FUNCTION_BLOCK MOTION_ACC_DCC
VAR_INPUT
	BOOL_UP_MOVE : BOOL;
	BOOL_DOWN_MOVE : BOOL;
	UINT_JOG_ACCDCC : UINT;
	UINT_HOME_ACCDCC : UINT;
	UINT_UD_ACCDCC : UINT;
	UINT_AG_ACCDCC : UINT;
	TIME_UD_DLY_ON : TIME;
	BOOL_MANUAL_PG : BOOL;
	BOOL_ORIGIN_COMP : BOOL;
	BOOL_ARM_HOME_READY : BOOL;
	STRING_CURRENT_PG : STRING;
	STRING_MAN_JOG_V_PG : STRING;
	STRING_MAN_POS_V_PG : STRING;
	STRING_MAN_JOG_H_PG : STRING;
	STRING_MAN_POS_H_PG : STRING;
END_VAR
VAR_OUTPUT

	UP_MOVE_ST_BOOL : BOOL;
	DOWN_MOVE_ST_BOOL : BOOL;
	ACC_UINT : UINT;
	DCC_UINT : UINT;

END_VAR
VAR
	T1: TON;
	T1COUNT: TIME;
	T2: TON;
	T2COUNT: TIME;
	MANJOGH: BOOL;
	MANJOGV: BOOL;
	MANPOSH: BOOL;
	MANPOSV: BOOL;
END_VAR
VAR // added by the converter: edge detectors and wires of the graphical bodies
    _w1, _w4, _w7, _w10 : BOOL;
    _w2, _w3, _w5, _w6, _w8, _w9, _w11, _w12 : UINT;
END_VAR

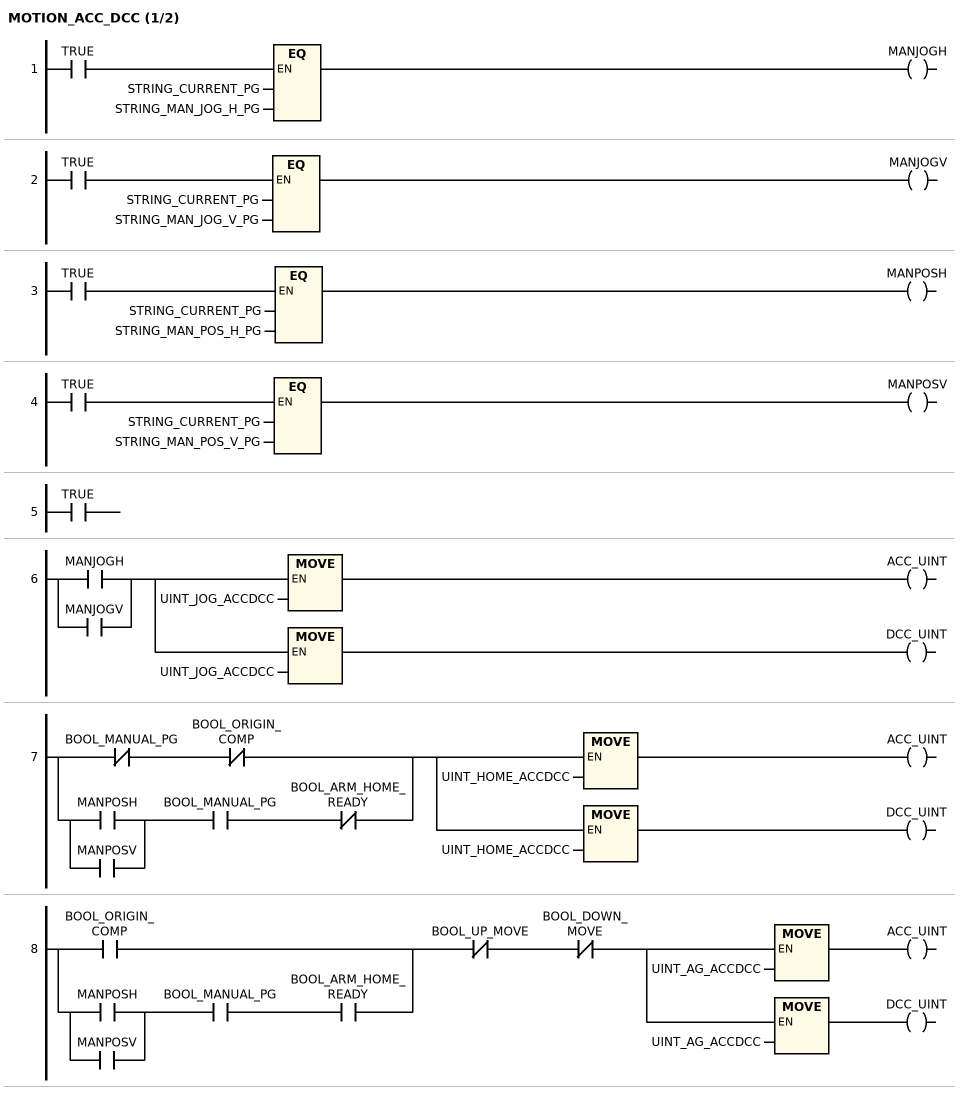
// NETWORK 1
MANJOGH := STRING_CURRENT_PG = STRING_MAN_JOG_H_PG;

// NETWORK 2
MANJOGV := STRING_CURRENT_PG = STRING_MAN_JOG_V_PG;

// NETWORK 3
MANPOSH := STRING_CURRENT_PG = STRING_MAN_POS_H_PG;

// NETWORK 4
MANPOSV := STRING_CURRENT_PG = STRING_MAN_POS_V_PG;

// NETWORK 5

// NETWORK 6
_w1 := MANJOGH OR MANJOGV;
IF _w1 THEN _w2 := UINT_JOG_ACCDCC; END_IF
ACC_UINT := _w2;
IF _w1 THEN _w3 := UINT_JOG_ACCDCC; END_IF
DCC_UINT := _w3;

// NETWORK 7
_w4 := NOT BOOL_MANUAL_PG AND NOT BOOL_ORIGIN_COMP OR (MANPOSH OR MANPOSV) AND BOOL_MANUAL_PG AND NOT BOOL_ARM_HOME_READY;
IF _w4 THEN _w5 := UINT_HOME_ACCDCC; END_IF
ACC_UINT := _w5;
IF _w4 THEN _w6 := UINT_HOME_ACCDCC; END_IF
DCC_UINT := _w6;

// NETWORK 8
_w7 := (BOOL_ORIGIN_COMP OR (MANPOSH OR MANPOSV) AND BOOL_MANUAL_PG AND BOOL_ARM_HOME_READY) AND NOT BOOL_UP_MOVE AND NOT BOOL_DOWN_MOVE;
IF _w7 THEN _w8 := UINT_AG_ACCDCC; END_IF
ACC_UINT := _w8;
IF _w7 THEN _w9 := UINT_AG_ACCDCC; END_IF
DCC_UINT := _w9;

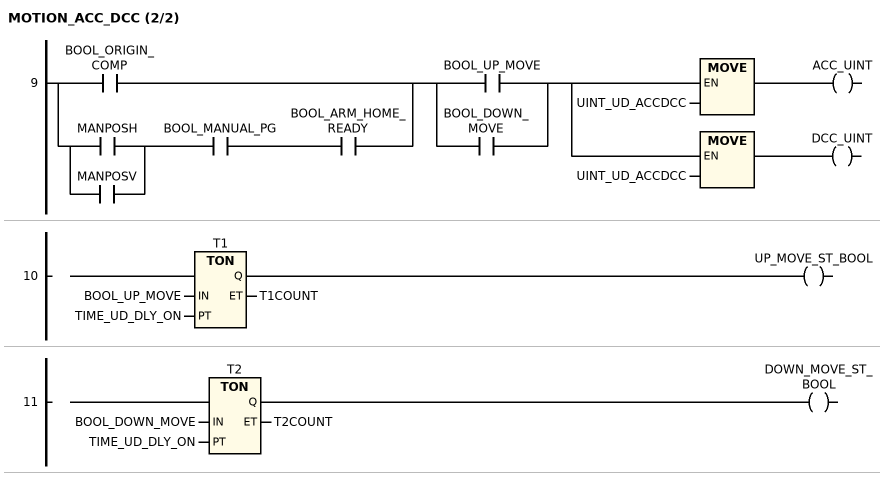
// NETWORK 9
_w10 := (BOOL_ORIGIN_COMP OR (MANPOSH OR MANPOSV) AND BOOL_MANUAL_PG AND BOOL_ARM_HOME_READY) AND (BOOL_UP_MOVE OR BOOL_DOWN_MOVE);
IF _w10 THEN _w11 := UINT_UD_ACCDCC; END_IF
ACC_UINT := _w11;
IF _w10 THEN _w12 := UINT_UD_ACCDCC; END_IF
DCC_UINT := _w12;

// NETWORK 10
T1(IN := BOOL_UP_MOVE, PT := TIME_UD_DLY_ON, ET => T1COUNT); // TON
UP_MOVE_ST_BOOL := T1.Q;

// NETWORK 11
T2(IN := BOOL_DOWN_MOVE, PT := TIME_UD_DLY_ON, ET => T2COUNT); // TON
DOWN_MOVE_ST_BOOL := T2.Q;

END_FUNCTION_BLOCK

(* stored: Version 1.1.0.1, ProductVersion 3.1.4024.12
   POU MOTION_ACC_DCC: Id {bf239d66-bbf8-4c74-92a6-1c09e786de1e}, SpecialFunc None *)
